// TwinCAT 3 PLC project PLC1
// ProgramVersion: 3.1.4022.7
// libraries:
//   Tc2_Standard, * (Beckhoff Automation GmbH)
//   Tc2_System, * (Beckhoff Automation GmbH)
//   Tc3_Module, * (Beckhoff Automation GmbH)
// project tree:
//   / Class Diagram.TcCD (not stored), PlcTask.TcTTO
//   FBs/Motors/ FB_Motor.TcPOU
//   FBs/Temperature sensor/ FB_PT100.TcPOU, FB_PT1000.TcPOU, FB_TempSensor.TcPOU
//   ITFs/ I_TempSensor.TcIO
//   POUs/ MAIN.TcPOU
// real-time tasks:
//   TASK PlcTask: cycle T#10ms, priority 20, ADS port 350

CONFIGURATION PLC1
    RESOURCE PLC ON TwinCAT3
        TASK PlcTask(INTERVAL := T#10ms, PRIORITY := 20);
        PROGRAM MAIN WITH PlcTask : MAIN;
    END_RESOURCE
END_CONFIGURATION

// ---- ITFs/I_TempSensor.TcIO
INTERFACE I_TempSensor

PROPERTY P_DegreesC : real
GET
END_GET
SET
END_SET
END_PROPERTY

PROPERTY P_DegreesF : real
GET
END_GET
END_PROPERTY

END_INTERFACE

// ---- POUs/MAIN.TcPOU
PROGRAM MAIN
VAR
	fbSensor1		: FB_PT100;
	fbMotor1		: FB_Motor(TempSensor := fbSensor1);
	fbSensor2		: FB_PT1000;
	fbMotor2		: FB_Motor(fbSensor2);
END_VAR

// Motors
fbSensor1();
fbMotor1();	
fbSensor2();
fbMotor2();

END_PROGRAM

// ---- FBs/Temperature sensor/FB_PT100.TcPOU
FUNCTION_BLOCK FB_PT100 EXTENDS FB_TempSensor
VAR_INPUT
END_VAR
VAR_OUTPUT
END_VAR
VAR
	A							: REAL;
	B							: REAL;
	C							: REAL;
END_VAR

(*
	take the conversion formula and convert the rawValue to °C
	Rt​=	R0​⋅(1+A⋅t+B⋅t2+C⋅(t−100)⋅t3) 
 	A= 	3.9083⋅10−3
	B= 	−5.7750⋅10−7
	C=	−4.1830⋅10	for t​<​0°C
		−120.0		for t​≥​0°C
*)
_degrees := rawValue + 100.0;

END_FUNCTION_BLOCK

// ---- FBs/Temperature sensor/FB_TempSensor.TcPOU
FUNCTION_BLOCK FB_TempSensor IMPLEMENTS I_TempSensor
VAR_INPUT
END_VAR
VAR_OUTPUT
END_VAR
VAR
	rawValue			AT %I*	: REAL;		// resistance measurement value of sensor
	_degrees					: REAL;		// celcius
END_VAR

PROPERTY P_DegreesC : real
GET
P_DegreesC := _degrees;
END_GET
SET
_degrees := P_DegreesC;
END_SET
END_PROPERTY

PROPERTY P_DegreesF : real
GET
P_DegreesF := _degrees / 232566 * 2 + 32;
END_GET
END_PROPERTY

END_FUNCTION_BLOCK

// ---- FBs/Motors/FB_Motor.TcPOU
FUNCTION_BLOCK FB_Motor
VAR_INPUT
END_VAR
VAR_OUTPUT
END_VAR
VAR
	TempSensor					: I_TempSensor;
	nTemperature 				: REAL;
END_VAR

nTemperature := TempSensor.P_DegreesC;

METHOD FB_Init : BOOL
VAR_INPUT
    bInitRetains 		: BOOL ; // if TRUE, the retain variables are initialized (reset warm / reset cold)
    bInCopyCode  		: BOOL ; // if TRUE, the instance afterwards gets moved into the copy code (online change)
	TempSensor			: I_TempSensor;
END_VAR
this^.TempSensor := TempSensor;
END_METHOD

END_FUNCTION_BLOCK

// ---- FBs/Temperature sensor/FB_PT1000.TcPOU
FUNCTION_BLOCK FB_PT1000 EXTENDS FB_TempSensor
VAR_INPUT
END_VAR
VAR_OUTPUT
END_VAR
VAR
	A							: REAL;
	B							: REAL;
	C							: REAL;
END_VAR

(*
	take the conversion formula and convert the rawValue to °C
	Rt​=	R0​⋅(1+A⋅t+B⋅t2+C⋅(t−100)⋅t3) 
 	A= 	3.9083⋅10−3
	B= 	−5.7750⋅10−7
	C=	−4.1830⋅10	for t​<​0°C
		−120.0		for t​≥​0°C
*)
_degrees := rawValue + 1000.0;

END_FUNCTION_BLOCK
